{attribute 'linkalways'} 
{attribute 'no_explicit_call' := 'This FB is a CLASS and must be accessed using methods or properties'}
{attribute 'enable_dynamic_creation'}
FUNCTION_BLOCK Node_F_VN_PointToPointDistance_TcVnPoint2_REAL EXTENDS VisionNode
VAR
    aPoint1 : _TcVnPoint2_REAL;
    aPoint2 : _TcVnPoint2_REAL;
    fDistance : _LREAL(0.0);
    hrPrev : _HRESULT(S_OK);
	hresult : _HRESULT(S_OK);
END_VAR

METHOD PUBLIC  Clone : I_Node
VAR
	pNode : POINTER TO Node_F_VN_PointToPointDistance_TcVnPoint2_REAL;
END_VAR
pNode := __NEW(Node_F_VN_PointToPointDistance_TcVnPoint2_REAL);
Clone := pNode^;
END_METHOD

METHOD FB_init : BOOL
VAR_INPUT
	bInitRetains : BOOL; // if TRUE, the retain variables are initialized (warm start / cold start)
	bInCopyCode : BOOL;  // if TRUE, the instance afterwards gets moved into the copy code (online change)
END_VAR
AddInput('aPoint1', aPoint1);
AddInput('aPoint2', aPoint2);
AddInput('hrPrev', hrPrev);
AddOutput('fDistance', fDistance);
AddOutput('hresult',hresult);
END_METHOD

METHOD PROTECTED OnExecute
hresult.Value := F_VN_PointToPointDistance_TcVnPoint2_REAL(
    aPoint1 := aPoint1.Value,
    aPoint2 := aPoint2.Value,
    fDistance := fDistance.Value,
	hrPrev:= hrPrev.Value);
END_METHOD

METHOD PUBLIC PreExecutionCheck
VAR_INPUT
	Check : I_PreExecutionChecks;
END_VAR
END_METHOD

END_FUNCTION_BLOCK

(* stored: Version 1.1.0.1, ProductVersion 3.1.4024.15
   POU Node_F_VN_PointToPointDistance_TcVnPoint2_REAL: Id {6332f6de-d6ff-074e-01df-302db06e42fd}, SpecialFunc None
   Folder Constructor: Id {62c23a35-5784-0317-3ed9-bb098a3f9437}
   Method Clone: Id {327b6d7d-be65-0e5a-0165-ee49c4290af9}
   Method FB_init: Id {47a2425c-2a0b-0892-0880-f11c93c0a96a}
   Method OnExecute: Id {2422bfe8-b3c4-02cf-2e0a-296fa9dbb383}
   Method PreExecutionCheck: Id {638254d9-54df-0cff-0f3f-dc3fba80cfce} *)
